(* CODESYS project PiPlate_DAQC.library
   Company: Lennart
   DefaultNamespace: PiPlate_DAQC
   Title: PiPlate_DAQC
   Description: Library containing device support of PiPlate DAQC Digital
   Placeholder: PlaceholderTemplate
   Author: Lennart Albertsen
   Version: 1.2.0.0

Project tree, tasks and I/O mapping:
  libraries: IoDrvGPIO, * (3S - Smart Software Solutions GmbH); Raspberry Pi Peripherals, * (3S - Smart Software Solutions GmbH); IoStandard, * (System)
  global variables GCL_PiPlate_DAQC
  00000000-0000-0000-0000-000000000000|D:\CoDeSys\LibrariesV3\trunk\Intern\CAA\CAA Template\3.4.0.0 draft\Placeholder.xml
  00000000-0000-0000-0000-000000000000|D:\CoDeSys\LibrariesV3\trunk\Intern\CAA\CAA Template\3.2.0.3 draft\Prefix.pdf
  00000000-0000-0000-0000-000000000000|D:\CoDeSys\LibrariesV3\trunk\Intern\CAA\CAA Template\3.5.2.0 draft\Placeholder.xml
  function block PiPlate_DAQC [ST]: Initialize, BeforeWriteOutputs, AfterReadInputs, read8, write8
*)

// GCL_PiPlate_DAQC
VAR_GLOBAL CONSTANT
	//OUTPUT_PORT: USINT := 16#0D;
	//INPUT_PORT: USINT := 16#19;
	//IOCON: USINT := 0;
	//GPIOA: USINT := 16#14;
	//GPIOB: USINT := 16#13;
	//GPPUB: USINT := 16#0D;
	//IODIRA: USINT := 16#00;
	//IODIRB: USINT := 16#01;
DELAY_SETTLE_NS : UDINT := 40000; // 40us
DELAY_SETTLE_NSX : UDINT := 400000; // 400us
END_VAR

// PiPlate_DAQC
FUNCTION_BLOCK PiPlate_DAQC EXTENDS spi
VAR_INPUT
	DO1:BOOL; //Digital Output 1
	DO2:BOOL; //Digital Output 2
	DO3:BOOL; //Digital Output 3
	DO4:BOOL; //Digital Output 4
	DO5:BOOL; //Digital Output 5
	DO6:BOOL; //Digital Output 6
	DO7:BOOL; //Digital Output 7
	AO1:UINT; //Analog Output 1 Range: 0..1023
	AO2:UINT; //Analog Output 2 Range: 0..1023
END_VAR
VAR_OUTPUT
	DI1:BOOL; //Digital Input 1
	DI2:BOOL; //Digital Input 2
	DI3:BOOL; //Digital Input 3
	DI4:BOOL; //Digital Input 4
	DI5:BOOL; //Digital Input 5
	DI6:BOOL; //Digital Input 6
	DI7:BOOL; //Digital Input 7
	DI8:BOOL; //Digital Input 8
	AI1:UINT; //Analog Input 1 Range: 0..1023
	AI2:UINT; //Analog Input 2 Range: 0..1023
	AI3:UINT; //Analog Input 3 Range: 0..1023
	AI4:UINT; //Analog Input 4 Range: 0..1023
	AI5:UINT; //Analog Input 5 Range: 0..1023
	AI6:UINT; //Analog Input 6 Range: 0..1023
	AI7:UINT; //Analog Input 7 Range: 0..1023
	AI8:UINT; //Analog Input 8 Range: 0..1023
	OPR:BOOL; //Operational
END_VAR
VAR
	_byHardwareAddress: BYTE;
	BoardBaseAddress:BYTE :=8;
	BoardType:ARRAY [0..20] OF BYTE :=[0,0,0,0,80,105,45,80,108,97,116,101,32,68,65,81,67,0,0,0,0]; (*Pi-Plate DAQC*)
	digitalOut:BYTE;
	digitalIn:BYTE;
	byInDO:BYTE;
	vState:INT;
	IOStatusOK:BOOL := TRUE;
	vRecArray:ARRAY [0..20] OF BYTE;
	PWMArray:ARRAY  [0..2] OF BYTE;
END_VAR
VAR_TEMP
	i, k: INT;
END_VAR

SUPER^();

CASE _iState OF
0:	IF SUPER^.init() THEN
		read8(_byHardwareAddress,00,0,0,1); //Check Control Board Address
		IF vRecArray[4] = _byHardwareAddress + BoardBaseAddress THEN
			read8(_byHardwareAddress,01,0,0,1); //Check Control Board Type
			IF vRecArray[4] = BoardType[4] AND vRecArray[5] = BoardType[5] AND vRecArray[6] = BoardType[6] AND vRecArray[7] = BoardType[7] AND vRecArray[8] = BoardType[8] AND vRecArray[9] = BoardType[9] AND vRecArray[10] = BoardType[10] AND vRecArray[11] = BoardType[11] AND vRecArray[12] = BoardType[12] AND vRecArray[13] = BoardType[13] AND vRecArray[14] = BoardType[14] AND vRecArray[15] = BoardType[15] AND vRecArray[16] = BoardType[16] AND vRecArray[17] = BoardType[17] THEN
				_iState := 1;
			END_IF
		END_IF;
	END_IF	
1: 	_iState := 10;

10: //Board Present an OK
	IF _pConnector^.dwFlags = 242 OR NOT IOStatusOK THEN
	_iState:=1000;
	END_IF
1000: _iState:=0;
END_CASE
OPR := Operational AND _iState = 10;
IF AO1 >= 1023 THEN
	AO1 := 1023;
END_IF;
IF AO2 >= 1023 THEN
	AO2 := 1023;
END_IF;

METHOD Initialize : UDINT
VAR_INPUT
	wModuleType : UINT;
	dwInstance : UDINT;
	pConnector : POINTER TO IoConfigConnector;
END_VAR
VAR
	pParam: POINTER TO IoConfigParameter;		
	udiResult: UDINT;
END_VAR
SUPER^.Initialize(wModuleType, dwInstance, pConnector);

pParam := ConfigGetParameter(_pConnector, 1);
IF pParam <> 0 THEN
	_byHardwareAddress := IoStandard.ConfigGetParameterValueByte(pParam, ADR(udiResult));
END_IF
END_METHOD

METHOD BeforeWriteOutputs : INT
VAR
	i: INT;
END_VAR
SUPER^.BeforeWriteOutputs();

IF _iState = 10 THEN
(*	
				digitalOut.0 := DO1;
				digitalOut.1 := DO2;	
				digitalOut.2 := DO3;
				digitalOut.3 := DO4;
				digitalOut.4 := DO5;
				digitalOut.5 := DO6;
				digitalOut.6 := DO7;
write8(_byHardwareAddress,19,digitalout,0,0); //Write Digital Outputs
				
				PWMArray[0] := UINT_TO_BYTE(AO1 /256);
				PWMArray[1] := UINT_TO_BYTE(AO1);
write8(_byHardwareAddress,64,PWMArray[0],PWMArray[1],0); //write Analog Out1/PWM

				PWMArray[0] := UINT_TO_BYTE(AO2 /256);
				PWMArray[1] := UINT_TO_BYTE(AO2);
write8(_byHardwareAddress,65,PWMArray[0],PWMArray[1],0); //write Analog Out1/PWM
END_IF *)
(* The CASE executes faster, code her and in AfterReadInputs are disabled*)

		CASE vState OF
	
			0: 	read8(_byHardwareAddress,37,0,0,1); // Get Digital Inputs
				digitalIn := NOT vRecArray[4]; // DI inputs status
				DI1 := digitalIn.0;
				DI2 := digitalIn.1;
				DI3 := digitalIn.2;
				DI4 := digitalIn.3;
				DI5 := digitalIn.4;
				DI6 := digitalIn.5;
				DI7 := digitalIn.6;
				DI8 := digitalIn.7;
				vState := 1;	
		
			1: 	digitalOut.0 := DO1;
				digitalOut.1 := DO2;	
				digitalOut.2 := DO3;
				digitalOut.3 := DO4;
				digitalOut.4 := DO5;
				digitalOut.5 := DO6;
				digitalOut.6 := DO7;
				write8(_byHardwareAddress,19,digitalout,0,0); //Write Digital Outputs
				vState := 2;
				
			2: 	read8(_byHardwareAddress,20,0,0,1); // Get Digital Output status
				byInDO := vRecArray[4]; //DO's status feedback
				IOStatusOK := byInDO = digitalout;
				vState := 3;
		
			3: 	read8(_byHardwareAddress,49,1,0,16); // Get Analog Inputs
				AI1 := 256*vRecArray[4]+vRecArray[5]; //AI1 calc 0..1024
				AI2 := 256*vRecArray[6]+vRecArray[7]; //AI2 calc 0..1024
				AI3 := 256*vRecArray[8]+vRecArray[9]; //AI3 calc 0..1024
				AI4 := 256*vRecArray[10]+vRecArray[11]; //AI4 calc 0..1024
				AI5 := 256*vRecArray[12]+vRecArray[13]; //AI5 calc 0..1024
				AI6 := 256*vRecArray[14]+vRecArray[15]; //AI6 calc 0..1024
				AI7 := 256*vRecArray[16]+vRecArray[17]; //AI7 calc 0..1024
				AI8 := 256*vRecArray[18]+vRecArray[19]; //AI8 calc 0..1024
				vState := 4;
		
			4:	PWMArray[0] := UINT_TO_BYTE(AO1 /256);
				PWMArray[1] := UINT_TO_BYTE(AO1);
				write8(_byHardwareAddress,64,PWMArray[0],PWMArray[1],0); //write Analog Out1/PWM
				vState := 5;
		
			5:	PWMArray[0] := UINT_TO_BYTE(AO2 /256);
				PWMArray[1] := UINT_TO_BYTE(AO2);
				write8(_byHardwareAddress,65,PWMArray[0],PWMArray[1],0); //write Analog Out1/PWM
				vState := 0;
		END_CASE
END_IF
END_METHOD

METHOD AfterReadInputs : INT
VAR
END_VAR
SUPER^.AfterReadInputs();
(*
IF _iState = 10 THEN
read8(_byHardwareAddress,37,0,0,1); // Get Digital Inputs
				digitalIn := NOT vRecArray[4]; // DI inputs status
				DI1 := digitalIn.0;
				DI2 := digitalIn.1;
				DI3 := digitalIn.2;
				DI4 := digitalIn.3;
				DI5 := digitalIn.4;
				DI6 := digitalIn.5;
				DI7 := digitalIn.6;
				DI8 := digitalIn.7;
				
read8(_byHardwareAddress,20,0,0,1); // Get Digital Output status
				byInDO := vRecArray[4]; //DO's status feedback
				IOStatusOK := byInDO = digitalout;
				
read8(_byHardwareAddress,49,1,0,16); // Get Analog Inputs
				AI1 := 256*vRecArray[4]+vRecArray[5]; //AI1 calc 0..1024
				AI2 := 256*vRecArray[6]+vRecArray[7]; //AI2 calc 0..1024
				AI3 := 256*vRecArray[8]+vRecArray[9]; //AI3 calc 0..1024
				AI4 := 256*vRecArray[10]+vRecArray[11]; //AI4 calc 0..1024
				AI5 := 256*vRecArray[12]+vRecArray[13]; //AI5 calc 0..1024
				AI6 := 256*vRecArray[14]+vRecArray[15]; //AI6 calc 0..1024
				AI7 := 256*vRecArray[16]+vRecArray[17]; //AI7 calc 0..1024
				AI8 := 256*vRecArray[18]+vRecArray[19]; //AI8 calc 0..1024
END_IF
*)
(*execution is faster with CASE in BeforeWriteOutputs *)
END_METHOD

// This method is used to read the data byte of one port using the following protocol:
// Byte0: hardware address + 8
// Byte1: Command
// Byte2: Parameter1
// Byte3: Parameter2
// Bytes to return are written to vRecArray
METHOD read8 : BYTE
VAR_INPUT
	byHardwareAddress: BYTE (0..7); (* hardware address *)
	CMD : BYTE;
	PARAM1 : BYTE;
	PARAM2 : BYTE;
	Bytes2return:BYTE;
END_VAR
VAR
	abyTxBuffer: ARRAY [0..3] OF BYTE;
	abyRxBuffer: ARRAY [0..20] OF BYTE;
	i:INT;
END_VAR
abyTxBuffer[0] := byHardwareAddress +8; //SPI_WRITE_CMD;
abyTxBuffer[1] := CMD;
abyTxBuffer[2] := PARAM1;
abyTxBuffer[3] := PARAM2;


IF bytes2return > 0 THEN
	IF transferExt(pabyTxBuffer:=ADR(abyTxBuffer) , pabyRxBuffer:=ADR(abyRxBuffer) , udiSpeedHz:=25000 , udiLen:=20 , uiDelayus:=5) THEN
		vRecArray := abyRxBuffer;
	ELSE
	_iState := 1000;	
	END_IF 
END_IF
END_METHOD

// This method is used to write a data byte into a port using the following protocol:
// Byte0: hardware address + 8
// Byte1: Command
// Byte2: Parameter1
// Byte3: Parameter2
// Bytes to return (not used here)
METHOD write8 : BOOL
VAR_INPUT
	byHardwareAddress: BYTE (0..7); (* hardware address *)
	CMD : BYTE;
	PARAM1 : BYTE;
	PARAM2 : BYTE;
	Bytes2return:BYTE;
	
END_VAR
VAR_OUTPUT
	
END_VAR
VAR
	abyTxBuffer: ARRAY [0..3] OF BYTE;
	abyRxTBuffer: ARRAY [0..20] OF BYTE;
	i:INT;
	y:DWORD;
END_VAR
abyTxBuffer[0] := byHardwareAddress +8; //SPI_WRITE_CMD;
abyTxBuffer[1] := CMD;
abyTxBuffer[2] := PARAM1;
abyTxBuffer[3] := PARAM2;
	
write8 := transferExt(pabyTxBuffer:=ADR(abyTxBuffer) , pabyRxBuffer:=ADR(abyRxTBuffer) , udiSpeedHz:=500000 , udiLen:=4 , uiDelayus:=1);

IF NOT write8 THEN
   _iState := 1000;
END_IF
END_METHOD

END_FUNCTION_BLOCK
